FUNCTION_BLOCK TExampleInterfaceImplementation IMPLEMENTS IExampleInterface
VAR_INPUT
END_VAR
VAR_OUTPUT
END_VAR
VAR
END_VAR

END_FUNCTION_BLOCK

(* stored: Version 1.1.0.1, ProductVersion 3.1.4024.4
   POU TExampleInterfaceImplementation: Id {67292391-722e-466e-b7ea-d2f4f341d700}, SpecialFunc None *)
